FUNCTION_BLOCK FB_Sequence
VAR_INPUT
	InStart:BOOL;
END_VAR
VAR_OUTPUT
	OutSequnceState:EN_SequenceState;
END_VAR
VAR
END_VAR

END_FUNCTION_BLOCK

(* stored: Version 1.1.0.1, ProductVersion 3.1.0.36
   POU FB_Sequence: Id {fb4892fb-69c3-469d-b6eb-dfd06ca281dc}, SpecialFunc None *)
